// TIA Portal V17 export
// export: Created 2025-03-05T08:02:47.6563183Z, ExportSetting WithDefaults, DisplayName Totally Integrated Automation Portal, DisplayVersion V17 Update 8, DisplayName TIA Portal Openness, DisplayVersion V17 Update 8, DisplayName TIA Portal Version Control Interface, DisplayVersion V17, DisplayName SINAMICS Startdrive Advanced, DisplayVersion V17 SP2, DisplayName SINAMICS Startdrive G110M, G120, G120C, G120D, G120P, G115D, DisplayVersion V17 SP2, DisplayName SINAMICS Startdrive G130, G150, S120, S150, SINAMICS MV, S210, DisplayVersion V17 SP2, DisplayName STEP 7 Professional, DisplayVersion V17 Update 8, DisplayName SINUMERIK ONE STEP 7 Toolbox, DisplayVersion V17 Update 12, DisplayName SINUMERIK 840D sl STEP 7 Toolbox, DisplayVersion V17 Update 12, DisplayName STEP 7 Safety, DisplayVersion V17 Update 6, DisplayName WinCC Advanced, DisplayVersion V17 Update 8
FUNCTION "FC2140_HOPPERS_BUTTONS" : Void   // FC2140, LAD
{ S7_Optimized_Access := 'FALSE' }
AUTHOR : ETXETAR
VERSION : 1.0
// stored: AutoNumber false, IsIECCheckEnabled false, SetENOAutomatically false, UDAEnableTagReadback false
   VAR_TEMP
      O_BYTE_0 : Struct   // OPTIONS BYTE 0
         IPC : Bool;   // IPC OPTION
      END_STRUCT;
      TCU_INDEX_SEL : Int;
   END_VAR
   VAR CONSTANT
      FC_NUMBER : DInt := 2140;   // FC NUMBER
   END_VAR
   VAR_TEMP   // added for the SCL form of the ladder/FBD networks
      _w1 : Bool;
   END_VAR
BEGIN

REGION Network 1: OPTIONS
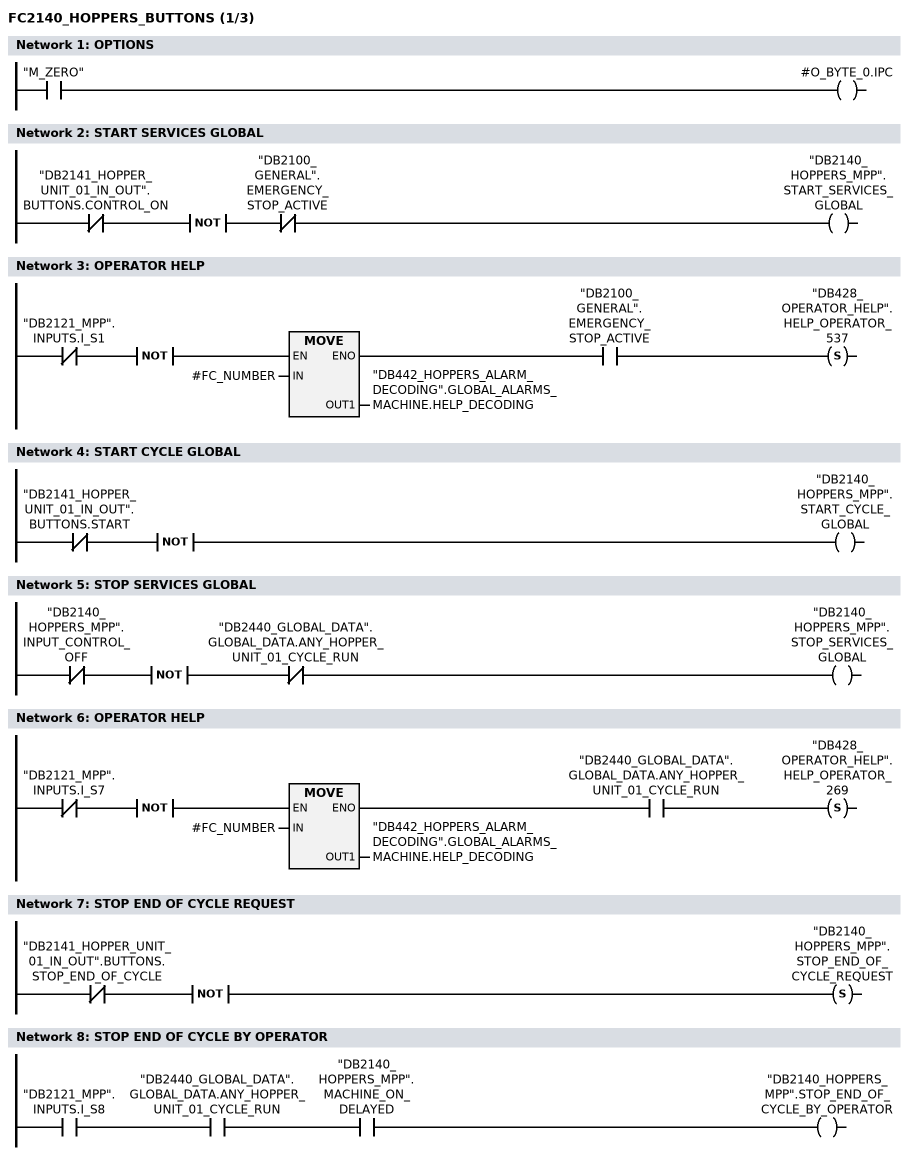
   RUNG wire#powerrail
      Contact( "M_ZERO" )
      Coil( #O_BYTE_0.IPC )
   END_RUNG
   // the same network as SCL:
   #O_BYTE_0.IPC := "M_ZERO";
END_REGION

REGION Network 2: START SERVICES GLOBAL
   RUNG wire#powerrail
      I_Contact( "DB2141_HOPPER_UNIT_01_IN_OUT".BUTTONS.CONTROL_ON )
      Not()
      I_Contact( "DB2100_GENERAL".EMERGENCY_STOP_ACTIVE )
      Coil( "DB2140_HOPPERS_MPP".START_SERVICES_GLOBAL )
   END_RUNG
   // the same network as SCL:
   "DB2140_HOPPERS_MPP".START_SERVICES_GLOBAL := NOT (NOT "DB2141_HOPPER_UNIT_01_IN_OUT".BUTTONS.CONTROL_ON) AND NOT "DB2100_GENERAL".EMERGENCY_STOP_ACTIVE;
END_REGION

REGION Network 3: OPERATOR HELP
   RUNG wire#powerrail
      I_Contact( "DB2121_MPP".INPUTS.I_S1 )
      Not()
      { S7_GenerateENO := "TRUE" } Move(in := #FC_NUMBER, out1 => "DB442_HOPPERS_ALARM_DECODING".GLOBAL_ALARMS_MACHINE.HELP_DECODING)
      Contact( "DB2100_GENERAL".EMERGENCY_STOP_ACTIVE )
      S_Coil( "DB428_OPERATOR_HELP".HELP_OPERATOR_537 )
   END_RUNG
   // the same network as SCL:
   // ENO of a box is taken as its EN; it also drops when the box reports an error
   #_w1 := NOT (NOT "DB2121_MPP".INPUTS.I_S1);
   IF #_w1 THEN "DB442_HOPPERS_ALARM_DECODING".GLOBAL_ALARMS_MACHINE.HELP_DECODING := #FC_NUMBER; END_IF;
   IF #_w1 AND "DB2100_GENERAL".EMERGENCY_STOP_ACTIVE THEN
       "DB428_OPERATOR_HELP".HELP_OPERATOR_537 := TRUE;
   END_IF;
END_REGION

REGION Network 4: START CYCLE GLOBAL
   RUNG wire#powerrail
      I_Contact( "DB2141_HOPPER_UNIT_01_IN_OUT".BUTTONS.START )
      Not()
      Coil( "DB2140_HOPPERS_MPP".START_CYCLE_GLOBAL )
   END_RUNG
   // the same network as SCL:
   "DB2140_HOPPERS_MPP".START_CYCLE_GLOBAL := NOT (NOT "DB2141_HOPPER_UNIT_01_IN_OUT".BUTTONS.START);
END_REGION

REGION Network 5: STOP SERVICES GLOBAL
   RUNG wire#powerrail
      I_Contact( "DB2140_HOPPERS_MPP".INPUT_CONTROL_OFF )
      Not()
      I_Contact( "DB2440_GLOBAL_DATA".GLOBAL_DATA.ANY_HOPPER_UNIT_01_CYCLE_RUN )
      Coil( "DB2140_HOPPERS_MPP".STOP_SERVICES_GLOBAL )
   END_RUNG
   // the same network as SCL:
   "DB2140_HOPPERS_MPP".STOP_SERVICES_GLOBAL := NOT (NOT "DB2140_HOPPERS_MPP".INPUT_CONTROL_OFF) AND NOT "DB2440_GLOBAL_DATA".GLOBAL_DATA.ANY_HOPPER_UNIT_01_CYCLE_RUN;
END_REGION

REGION Network 6: OPERATOR HELP
   RUNG wire#powerrail
      I_Contact( "DB2121_MPP".INPUTS.I_S7 )
      Not()
      { S7_GenerateENO := "TRUE" } Move(in := #FC_NUMBER, out1 => "DB442_HOPPERS_ALARM_DECODING".GLOBAL_ALARMS_MACHINE.HELP_DECODING)
      Contact( "DB2440_GLOBAL_DATA".GLOBAL_DATA.ANY_HOPPER_UNIT_01_CYCLE_RUN )
      S_Coil( "DB428_OPERATOR_HELP".HELP_OPERATOR_269 )
   END_RUNG
   // the same network as SCL:
   // ENO of a box is taken as its EN; it also drops when the box reports an error
   #_w1 := NOT (NOT "DB2121_MPP".INPUTS.I_S7);
   IF #_w1 THEN "DB442_HOPPERS_ALARM_DECODING".GLOBAL_ALARMS_MACHINE.HELP_DECODING := #FC_NUMBER; END_IF;
   IF #_w1 AND "DB2440_GLOBAL_DATA".GLOBAL_DATA.ANY_HOPPER_UNIT_01_CYCLE_RUN THEN
       "DB428_OPERATOR_HELP".HELP_OPERATOR_269 := TRUE;
   END_IF;
END_REGION

REGION Network 7: STOP END OF CYCLE REQUEST
   RUNG wire#powerrail
      I_Contact( "DB2141_HOPPER_UNIT_01_IN_OUT".BUTTONS.STOP_END_OF_CYCLE )
      Not()
      S_Coil( "DB2140_HOPPERS_MPP".STOP_END_OF_CYCLE_REQUEST )
   END_RUNG
   // the same network as SCL:
   IF NOT (NOT "DB2141_HOPPER_UNIT_01_IN_OUT".BUTTONS.STOP_END_OF_CYCLE) THEN
       "DB2140_HOPPERS_MPP".STOP_END_OF_CYCLE_REQUEST := TRUE;
   END_IF;
END_REGION

REGION Network 8: STOP END OF CYCLE BY OPERATOR
   RUNG wire#powerrail
      Contact( "DB2121_MPP".INPUTS.I_S8 )
      Contact( "DB2440_GLOBAL_DATA".GLOBAL_DATA.ANY_HOPPER_UNIT_01_CYCLE_RUN )
      Contact( "DB2140_HOPPERS_MPP".MACHINE_ON_DELAYED )
      Coil( "DB2140_HOPPERS_MPP".STOP_END_OF_CYCLE_BY_OPERATOR )
   END_RUNG
   // the same network as SCL:
   "DB2140_HOPPERS_MPP".STOP_END_OF_CYCLE_BY_OPERATOR := "DB2121_MPP".INPUTS.I_S8 AND "DB2440_GLOBAL_DATA".GLOBAL_DATA.ANY_HOPPER_UNIT_01_CYCLE_RUN AND "DB2140_HOPPERS_MPP".MACHINE_ON_DELAYED;
END_REGION

REGION Network 9: MAIN PANEL OPERATOR REQUEST STOP AT END OF CYCLE
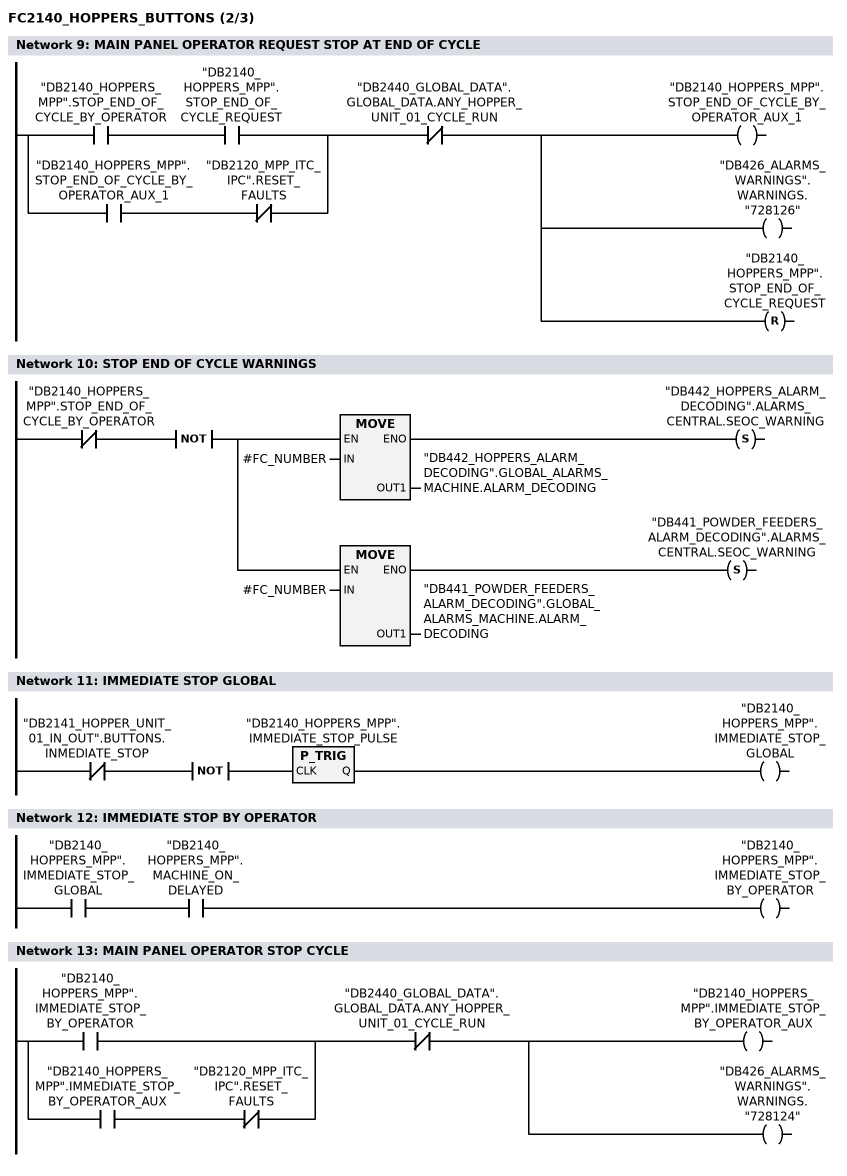
   RUNG wire#powerrail
      Contact( "DB2140_HOPPERS_MPP".STOP_END_OF_CYCLE_BY_OPERATOR )
      Contact( "DB2140_HOPPERS_MPP".STOP_END_OF_CYCLE_REQUEST )
      wire#w1
      I_Contact( "DB2440_GLOBAL_DATA".GLOBAL_DATA.ANY_HOPPER_UNIT_01_CYCLE_RUN )
      wire#w2
      Coil( "DB2140_HOPPERS_MPP".STOP_END_OF_CYCLE_BY_OPERATOR_AUX_1 )
   END_RUNG
   RUNG wire#powerrail
      Contact( "DB2140_HOPPERS_MPP".STOP_END_OF_CYCLE_BY_OPERATOR_AUX_1 )
      I_Contact( "DB2120_MPP_ITC_IPC".RESET_FAULTS )
   END_RUNG wire#w1
   RUNG wire#w2
      Coil( "DB426_ALARMS_WARNINGS".WARNINGS."728126" )
   END_RUNG
   RUNG wire#w2
      R_Coil( "DB2140_HOPPERS_MPP".STOP_END_OF_CYCLE_REQUEST )
   END_RUNG
   // the same network as SCL:
   "DB2140_HOPPERS_MPP".STOP_END_OF_CYCLE_BY_OPERATOR_AUX_1 := (("DB2140_HOPPERS_MPP".STOP_END_OF_CYCLE_BY_OPERATOR AND "DB2140_HOPPERS_MPP".STOP_END_OF_CYCLE_REQUEST) OR ("DB2140_HOPPERS_MPP".STOP_END_OF_CYCLE_BY_OPERATOR_AUX_1 AND NOT "DB2120_MPP_ITC_IPC".RESET_FAULTS)) AND NOT "DB2440_GLOBAL_DATA".GLOBAL_DATA.ANY_HOPPER_UNIT_01_CYCLE_RUN;
   "DB426_ALARMS_WARNINGS".WARNINGS."728126" := "DB2140_HOPPERS_MPP".STOP_END_OF_CYCLE_BY_OPERATOR_AUX_1;
   IF "DB2140_HOPPERS_MPP".STOP_END_OF_CYCLE_BY_OPERATOR_AUX_1 THEN
       "DB2140_HOPPERS_MPP".STOP_END_OF_CYCLE_REQUEST := FALSE;
   END_IF;
END_REGION

REGION Network 10: STOP END OF CYCLE WARNINGS
   RUNG wire#powerrail
      I_Contact( "DB2140_HOPPERS_MPP".STOP_END_OF_CYCLE_BY_OPERATOR )
      Not()
      wire#w1
      { S7_GenerateENO := "TRUE" } Move(in := #FC_NUMBER, out1 => "DB442_HOPPERS_ALARM_DECODING".GLOBAL_ALARMS_MACHINE.ALARM_DECODING)
      S_Coil( "DB442_HOPPERS_ALARM_DECODING".ALARMS_CENTRAL.SEOC_WARNING )
   END_RUNG
   RUNG wire#w1
      { S7_GenerateENO := "TRUE" } Move(in := #FC_NUMBER, out1 => "DB441_POWDER_FEEDERS_ALARM_DECODING".GLOBAL_ALARMS_MACHINE.ALARM_DECODING)
      S_Coil( "DB441_POWDER_FEEDERS_ALARM_DECODING".ALARMS_CENTRAL.SEOC_WARNING )
   END_RUNG
   // the same network as SCL:
   // ENO of a box is taken as its EN; it also drops when the box reports an error
   IF NOT (NOT "DB2140_HOPPERS_MPP".STOP_END_OF_CYCLE_BY_OPERATOR) THEN
       "DB442_HOPPERS_ALARM_DECODING".GLOBAL_ALARMS_MACHINE.ALARM_DECODING := #FC_NUMBER;
       "DB442_HOPPERS_ALARM_DECODING".ALARMS_CENTRAL.SEOC_WARNING := TRUE;
       "DB441_POWDER_FEEDERS_ALARM_DECODING".GLOBAL_ALARMS_MACHINE.ALARM_DECODING := #FC_NUMBER;
       "DB441_POWDER_FEEDERS_ALARM_DECODING".ALARMS_CENTRAL.SEOC_WARNING := TRUE;
   END_IF;
END_REGION

REGION Network 11: IMMEDIATE STOP GLOBAL
   RUNG wire#powerrail
      I_Contact( "DB2141_HOPPER_UNIT_01_IN_OUT".BUTTONS.INMEDIATE_STOP )
      Not()
      P_Trig( "DB2140_HOPPERS_MPP".IMMEDIATE_STOP_PULSE )
      Coil( "DB2140_HOPPERS_MPP".IMMEDIATE_STOP_GLOBAL )
   END_RUNG
   // the same network as SCL:
   #_w1 := NOT (NOT "DB2141_HOPPER_UNIT_01_IN_OUT".BUTTONS.INMEDIATE_STOP) AND NOT "DB2140_HOPPERS_MPP".IMMEDIATE_STOP_PULSE;   // rising edge
   "DB2140_HOPPERS_MPP".IMMEDIATE_STOP_PULSE := NOT (NOT "DB2141_HOPPER_UNIT_01_IN_OUT".BUTTONS.INMEDIATE_STOP);
   "DB2140_HOPPERS_MPP".IMMEDIATE_STOP_GLOBAL := #_w1;
END_REGION

REGION Network 12: IMMEDIATE STOP BY OPERATOR
   RUNG wire#powerrail
      Contact( "DB2140_HOPPERS_MPP".IMMEDIATE_STOP_GLOBAL )
      Contact( "DB2140_HOPPERS_MPP".MACHINE_ON_DELAYED )
      Coil( "DB2140_HOPPERS_MPP".IMMEDIATE_STOP_BY_OPERATOR )
   END_RUNG
   // the same network as SCL:
   "DB2140_HOPPERS_MPP".IMMEDIATE_STOP_BY_OPERATOR := "DB2140_HOPPERS_MPP".IMMEDIATE_STOP_GLOBAL AND "DB2140_HOPPERS_MPP".MACHINE_ON_DELAYED;
END_REGION

REGION Network 13: MAIN PANEL OPERATOR STOP CYCLE
   RUNG wire#powerrail
      Contact( "DB2140_HOPPERS_MPP".IMMEDIATE_STOP_BY_OPERATOR )
      wire#w1
      I_Contact( "DB2440_GLOBAL_DATA".GLOBAL_DATA.ANY_HOPPER_UNIT_01_CYCLE_RUN )
      wire#w2
      Coil( "DB2140_HOPPERS_MPP".IMMEDIATE_STOP_BY_OPERATOR_AUX )
   END_RUNG
   RUNG wire#powerrail
      Contact( "DB2140_HOPPERS_MPP".IMMEDIATE_STOP_BY_OPERATOR_AUX )
      I_Contact( "DB2120_MPP_ITC_IPC".RESET_FAULTS )
   END_RUNG wire#w1
   RUNG wire#w2
      Coil( "DB426_ALARMS_WARNINGS".WARNINGS."728124" )
   END_RUNG
   // the same network as SCL:
   "DB2140_HOPPERS_MPP".IMMEDIATE_STOP_BY_OPERATOR_AUX := ("DB2140_HOPPERS_MPP".IMMEDIATE_STOP_BY_OPERATOR OR ("DB2140_HOPPERS_MPP".IMMEDIATE_STOP_BY_OPERATOR_AUX AND NOT "DB2120_MPP_ITC_IPC".RESET_FAULTS)) AND NOT "DB2440_GLOBAL_DATA".GLOBAL_DATA.ANY_HOPPER_UNIT_01_CYCLE_RUN;
   "DB426_ALARMS_WARNINGS".WARNINGS."728124" := "DB2140_HOPPERS_MPP".IMMEDIATE_STOP_BY_OPERATOR_AUX;
END_REGION

REGION Network 14: IMMEDIATE STOP WARNING
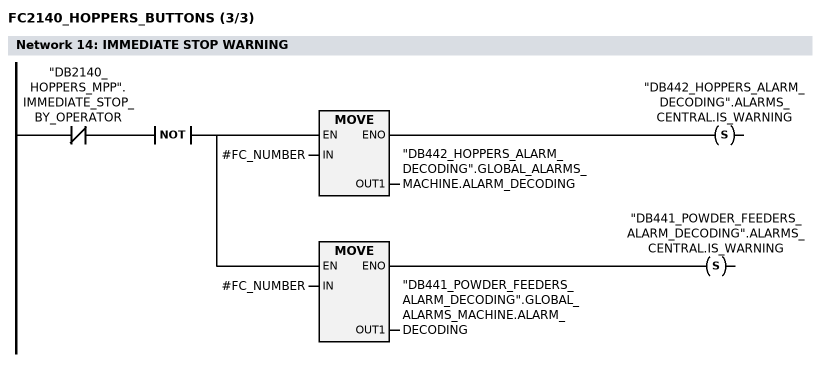
   RUNG wire#powerrail
      I_Contact( "DB2140_HOPPERS_MPP".IMMEDIATE_STOP_BY_OPERATOR )
      Not()
      wire#w1
      { S7_GenerateENO := "TRUE" } Move(in := #FC_NUMBER, out1 => "DB442_HOPPERS_ALARM_DECODING".GLOBAL_ALARMS_MACHINE.ALARM_DECODING)
      S_Coil( "DB442_HOPPERS_ALARM_DECODING".ALARMS_CENTRAL.IS_WARNING )
   END_RUNG
   RUNG wire#w1
      { S7_GenerateENO := "TRUE" } Move(in := #FC_NUMBER, out1 => "DB441_POWDER_FEEDERS_ALARM_DECODING".GLOBAL_ALARMS_MACHINE.ALARM_DECODING)
      S_Coil( "DB441_POWDER_FEEDERS_ALARM_DECODING".ALARMS_CENTRAL.IS_WARNING )
   END_RUNG
   // the same network as SCL:
   // ENO of a box is taken as its EN; it also drops when the box reports an error
   IF NOT (NOT "DB2140_HOPPERS_MPP".IMMEDIATE_STOP_BY_OPERATOR) THEN
       "DB442_HOPPERS_ALARM_DECODING".GLOBAL_ALARMS_MACHINE.ALARM_DECODING := #FC_NUMBER;
       "DB442_HOPPERS_ALARM_DECODING".ALARMS_CENTRAL.IS_WARNING := TRUE;
       "DB441_POWDER_FEEDERS_ALARM_DECODING".GLOBAL_ALARMS_MACHINE.ALARM_DECODING := #FC_NUMBER;
       "DB441_POWDER_FEEDERS_ALARM_DECODING".ALARMS_CENTRAL.IS_WARNING := TRUE;
   END_IF;
END_REGION
END_FUNCTION
